{attribute 'TcGenerated'}
{attribute 'no-analysis'}
{attribute 'linkalways'}
// This function has been automatically generated from the project information.
VAR_GLOBAL CONSTANT
	{attribute 'const_non_replaced'}
	stLibVersion_PDxx : ST_LibVersion := (iMajor := 0, iMinor := 3, iBuild := 2, iRevision := 0, nFlags := 1, sVersion := '0.3.2.0');
END_VAR

(* stored: Version 1.1.0.1, ProductVersion 3.1.4024.15
   GVL Global_Version: Id {53ae8b4c-8f21-4d21-8297-85127d0403a6} *)
